// Mitsubishi GX Works2 project: z03   PLC: Q02/Q02H

PROGRAM MAIN
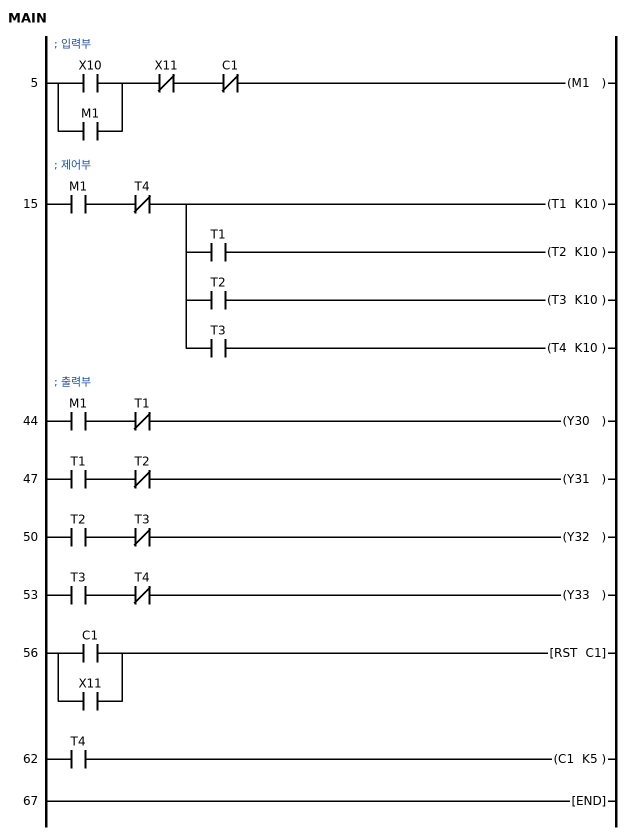
; 입력부
5     LD      X10
      OR      M1
      ANI     X11
      ANI     C1
      OUT     M1
; 제어부
15    LD      M1
      ANI     T4
      OUT     T1 K10
      MPS
      AND     T1
      OUT     T2 K10
      MRD
      AND     T2
      OUT     T3 K10
      MPP
      AND     T3
      OUT     T4 K10
; 출력부
44    LD      M1
      ANI     T1
      OUT     Y30
47    LD      T1
      ANI     T2
      OUT     Y31
50    LD      T2
      ANI     T3
      OUT     Y32
53    LD      T3
      ANI     T4
      OUT     Y33
56    LD      C1
      OR      X11
      RST     C1
62    LD      T4
      OUT     C1 K5
67    END
END_PROGRAM
